Yaskawa INFORM job: PP1.JBI

/JOB
//NAME PP1
///FOLDERNAME FOLDER001
//POS
///NPOS 0,0,0,5,0,0
///TOOL 0
///POSTYPE PULSE
///PULSE
P00001=55242,26922,11446,1601,-60437,64378
P00002=55242,35623,-7881,1830,-43902,63991
P00004=-47424,25138,-17957,938,-40698,102661
P00005=56012,31125,28227,2771,-69762,62996
P00006=-50960,20794,17892,682,-65721,104273
//INST
///DATE 2025/12/05 13:12
///ATTR SC,RW
///GROUP1 RB1
NOP
DOUT OT#(9) ON
MOVJ P001 VJ=20.00 PL=0
MOVL P002 V=80.0 PL=0
TIMER T=0.300
DOUT OT#(10) ON
TIMER T=0.500
MOVL P001 V=80.0 PL=0
MOVJ P006 VJ=20.00 PL=0
MOVL P004 V=80.0 PL=0
TIMER T=0.300
DOUT OT#(10) OFF
TIMER T=0.500
MOVL P006 V=80.0 PL=0
DOUT OT#(9) OFF
END
